// TIA Portal V19 export
DATA_BLOCK "PNIO_Diagnostic_Data"   // DB17
TITLE = Data for PNIODiagnostics
{ S7_Optimized_Access := 'TRUE' }
AUTHOR : NDJH
// stored: MemoryReserve 100
   VAR
      "2_AL1103" : "DiagnosticUDT";
      "3_AL1307" : "DiagnosticUDT";
      "4_AL1307" : "DiagnosticUDT";
      "5_AL1307" : "DiagnosticUDT";
      "6_AL1307" : "DiagnosticUDT";
      "7_AL1307" : "DiagnosticUDT";
      "8_Promag300" : "DiagnosticUDT";
      "9_SinaG120" : "DiagnosticUDT";
      "10_AL1307" : "DiagnosticUDT";
      "11_PNCoup" : "DiagnosticUDT";
      "12_AL1307" : "DiagnosticUDT";
      "2_AL1103_Historical" : "DiagnosticUDT";
      "3_AL1307_Historical" : "DiagnosticUDT";
      "4_AL1307_Historical" : "DiagnosticUDT";
      "5_AL1307_Historical" : "DiagnosticUDT";
      "6_AL1307_Historical" : "DiagnosticUDT";
      "7_AL1307_Historical" : "DiagnosticUDT";
      "8_Promag300_Historical" : "DiagnosticUDT";
      "9_SinaG120_Historical" : "DiagnosticUDT";
      "10_AL1307_Historical" : "DiagnosticUDT";
      "11_PNCoup_Historical" : "DiagnosticUDT";
      "12_AL1307_Historical" : "DiagnosticUDT";
   END_VAR
BEGIN
END_DATA_BLOCK
